{attribute 'strict'}
TYPE E_GoldenSampleMeasurementState :
(
	GOLDEN_SAMPLE_MEASUREMENT_IDLE 									:= 0,
	
	GOLDEN_SAMPLE_MEASUREMENT_ROBOT_GO_TO_SAMPLE					:= 40,
	GOLDEN_SAMPLE_MEASUREMENT_ROBOT_PICK_SAMPLE						:= 50,
	
	GOLDEN_SAMPLE_MEASUREMENT_ROBOT_GO_TO_STATION_1					:= 60,
	GOLDEN_SAMPLE_MEASUREMENT_ROBOT_GO_TO_STATION_1_DONE			:= 70,
	GOLDEN_SAMPLE_MEASUREMENT_ROBOT_GO_TO_STATION_2					:= 80,
	GOLDEN_SAMPLE_MEASUREMENT_ROBOT_GO_TO_STATION_2_DONE			:= 90,
	
	GOLDEN_SAMPLE_MEASUREMENT_ROBOT_GO_TO_REJECTBOX					:= 100,
	GOLDEN_SAMPLE_MEASUREMENT_ROBOT_GO_TO_ROTARY_TABLE				:= 110,
	GOLDEN_SAMPLE_MEASUREMENT_ROBOT_DROP_PRODUCT_ROTARY_TABLE		:= 115,
	GOLDEN_SAMPLE_MEASUREMENT_ROBOT_DROP_PRODUCT_ROTARY_TABLE_DONE	:= 120,
	
	GOLDEN_SAMPLE_MEASUREMENT_ROBOT_GO_TO_OUT_POSITION				:= 130,
	GOLDEN_SAMPLE_MEASUREMENT_ROBOT_GO_TO_OUT_POSITION_PICK			:= 135,
		
	GOLDEN_SAMPLE_MEASUREMENT_ROBOT_RETURN_TO_STATION				:= 140,
	GOLDEN_SAMPLE_MEASUREMENT_ROBOT_RETURN_TO_STATION_PLACED		:= 150,
	GOLDEN_SAMPLE_MEASUREMENT_ROBOT_RETURN_TO_STATION_PLACED_DONE	:= 160,
	
	GOLDEN_SAMPLE_MEASUREMENT_CHECK_RESULTS							:= 180,
	
	GOLDEN_SAMPLE_MEASUREMENT_GO_SAFE_POSITION						:= 190,
	GOLDEN_SAMPLE_MEASUREMENT_SAFE_POSITION_DONE					:= 200,
	
	GOLDEN_SAMPLE_MEASUREMENT_OK 									:= 210,
	GOLDEN_SAMPLE_MEASUREMENT_FAIL 									:= 220,
	GOLDEN_SAMPLE_MEASUREMENT_STOPPED								:= 230
);
END_TYPE

(* stored: Version 1.1.0.1, ProductVersion 3.1.4024.9
   DUT E_GoldenSampleMeasurementState: Id {a31e52e7-c884-4540-a704-0194e3284f04} *)
